{attribute addProperty BoxType "EL3102--0000"}
{attribute addProperty Id "ChannelAT %I*ARRAY[0..1] OF Channel_A23A2BD94860WcStateAT %I*WcState_F855686C1620InfoDataAT %I*InfoData_BC63D37F80100"}
{attribute addProperty CRC "845178501"}
{attribute addProperty SizeInBites "144"}
{attribute addProperty SizeInBytes "18"}
TYPE EL3102_B73BDD58 :
STRUCT
	{attribute addProperty Name "Channel"}
	Channel : ARRAY[0..1] OF Channel_A23A2BD9;
	{attribute addProperty Name "WcState"}
	WcState : WcState_F855686C;
	{attribute addProperty Name "InfoData"}
	InfoData : InfoData_BC63D37F;
END_STRUCT
END_TYPE

(* stored: Version 1.2.0.0, ProductVersion 3.1.4024.9
   DUT EL3102_B73BDD58: Id {1d5909a9-d23b-469d-bfb4-aae65480afa3} *)
